// TIA Portal V16 export
// export: Created 2023-03-29T11:04:30.0002099Z, ExportSetting WithDefaults, DisplayName Totally Integrated Automation Portal, DisplayVersion V16 Update 6, DisplayName TIA Portal Version Control Interface, DisplayVersion V16 Update 2, DisplayName TIA Portal Openness, DisplayVersion V16 Update 6, DisplayName STEP 7 Professional, DisplayVersion V16 Update 6, DisplayName STEP 7 Safety, DisplayVersion V16, DisplayName WinCC Advanced, DisplayVersion V16 Update 6
DATA_BLOCK "Dane_ComunicationControlHMI"   // DB29
TITLE = WatchDog HMI-Krata - S7-Krata
{ S7_Optimized_Access := 'FALSE' }
AUTHOR : rtecmer
VERSION : 0.1
// stored: AutoNumber true, DBAccessibleFromOPCUA true, IsOnlyStoredInLoadMemory false, IsWriteProtectedInAS false
   VAR
      Data_czas_loc : DTL;   // Zegar dla panelu HMI Krata
      WatchDog_WinCC : Word;   // Zmienna kordynująca kontrolę komunikacji od strony PC WinCC.
      SetFaultComunikation_Zasuwy : Int;   // Kontrola komunikacji z HMI
      Data_czas_sys : DTL;   // Zegar dla panelu HMI Krata
      Data_czasHMI : DTL;   // Zegar czytany z funkcji RTC (FC44) zapas
      tempCoordinationHMIRS5 : Int;   // Kontrola CoorditionHMI KDN
      tempWatchDog_WinCC : Word;   // Zmienna kordynująca kontrolę komunikacji od strony PC WinCC.
   END_VAR
BEGIN
END_DATA_BLOCK
